FUNCTION_BLOCK FB_ConvStatistic
VAR_INPUT
    // Time to be written into the ring buffer
    tLapTime : TIME;
    bAddValue : BOOL;
END_VAR
VAR_OUTPUT
	// Last 10 lap times
	aLapTimes: ARRAY[0..10] OF TIME;
END_VAR
VAR
    // Current index of array
    nIndex : INT := 1;
	bAddValueIsset: BOOL;
END_VAR

IF bAddValue AND NOT bAddValueIsset THEN
    aLapTimes[nIndex] := tLapTime;

    IF nIndex >= 10 THEN
        nIndex := 1;
    ELSE
        nIndex := nIndex + 1;
    END_IF
END_IF

bAddValueIsset := bAddValue;

END_FUNCTION_BLOCK

(* stored: Version 1.1.0.1
   POU FB_ConvStatistic: Id {f93cda1a-379b-43cf-a2b0-159c80785fe5}, SpecialFunc None *)
